# B&R Automation Studio project LMS47
Automation Studio 4.2.7.54 SP

## Configuration Config2

CPU 5PPC2100.BY22-000, AutomationRuntime B4.26, Build 4.1.2, Vc V4.26.2, Safety 0.0

### Task classes (Cpu.sw)
```
NcDataObjects: acp10etxen <- acp10etxen.dob, gAxis01i <- gAxis01obj.gAxis01i.dob, LMS47Liden <- gAxis01obj.LMS47Liden.dob
Libraries: Acp10man, Acp10par, NcGlobal, Acp10_MC, brsystem, sys_lib, runtime
```

### Hardware
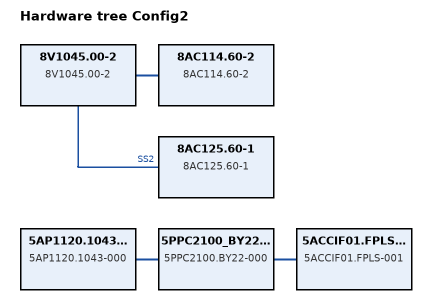
```
5ACCIF01.FPLS-001 : 5ACCIF01.FPLS-001 v1.2.0.0  [SL -> 5PPC2100_BY22_000b.SL1]
5AP1120.1043-000 : 5AP1120.1043-000 v1.0.1.0
5PPC2100_BY22_000b : 5PPC2100.BY22-000 v1.2.4.0  [SY -> 5AP1120.1043-000.SY1]
  Connector IF3:
    ActivateDevice = 1
  Connector IF4:
    ActivateDevice = 1
    Mode = Manual
    InternetAddress = 192.168.0.13
    SubnetMask = 255.255.255.0
  ConfigurationID = LMS47_Config2
  TimerDeviceType = EPLX2X
  TaskClassIdleTime = 2000
  Cyclic1Duration = 2000
  Cyclic1Tolerance = 0
  Cyclic2Duration = 20000
  Cyclic2Tolerance = 20000
  Cyclic3Duration = 50000
  Cyclic3Tolerance = 50000
  Cyclic4Duration = 100000
  Cyclic4Tolerance = 100000
  Cyclic5Duration = 200000
  Cyclic5Tolerance = 200000
  Cyclic6Duration = 500000
  Cyclic6Tolerance = 500000
  Cyclic7Duration = 1000000
  Cyclic7Tolerance = 1000000
  Cyclic8Duration = 10000
  Cyclic8Tolerance = 30000000
  TimerDevice = 5ACCIF01.FPLS-001.IF1
8AC114.60-2 : 8AC114.60-2 v1.0.0.8  [SS -> 8V1045.00-2.SS1; PLK1 -> 5ACCIF01.FPLS-001.IF1 (NodeNumber=1)]
8AC125.60-1 : 8AC125.60-1 v1.0.0.2  [SS -> 8V1045.00-2.SS2]
8V1045.00-2 : 8V1045.00-2 v1.0.0.2
  QuickStopIsNormallyOpen_r1 = on
```

### Acp10cfg.ncc - 5PPC2100_BY22_000b/Motion/Acp10cfg.ncc
```
NcConfiguration (Version=3.15.1, NcSwId=Acp10)
  ACP10CF1_typ:
    cnt_nettrc_rec_drive = 1500
    bufsize_trace_upload = 1200
    tc_nc_man_task = Cyclic #1
    glob_pv_as_ncobject = Yes
    ncsys_dl_broadcast = Yes
    ncsys_dl_acp_reset = Yes
    safemc_log_err_to_ax = Yes
    network_init:
      ncsw_init_execute = Yes
      automatic_execute = No
      node_nr_warning = Yes
      net_err_before_ncact = Yes
    nettrc:
      enter_parsecrec = Yes
      enter_ncaction = Yes
      save_ring_startidx = Yes
    cam_prof_download:
      cam_dat_dl_parallel = No
      tc_cam_dl_parallel = Task class for NC Manager task
    plk_if[0]:
      if_name = SL1.SS1.IF2
      tc_CycDat_PLCopen = Task class for NC Manager task
      mc_broadcast_extdat = No
    plk_if[1]:
      if_name = IF1
      tc_CycDat_PLCopen = Task class for NC Manager task
      mc_broadcast_extdat = No
    plk_if[2]:
      if_name = SL1.IF2
      tc_CycDat_PLCopen = Task class for NC Manager task
      mc_broadcast_extdat = No
    plk_if[3]:
      if_name = SL1.IF1
      tc_CycDat_PLCopen = Task class for NC Manager task
      mc_broadcast_extdat = No
```

### Acp10map.ncm - 5PPC2100_BY22_000b/Motion/Acp10map.ncm
```
NcMapping (NcSwId=Acp10, DisabledNodesAreHidden=False)
  NcObject gAxis01 (ModuleId=8V1045.00-2, Type=ncAXIS, Channel=1, AcoposSimulation=Off, InitParameter=gAxis01i, AcoposParameter=LMS47Liden, Disabled=FALSE, ModuleDisabled=FALSE)
  NcObject 8V1045.00-2_ncV_AXIS1 (ModuleId=8V1045.00-2, Type=ncV_AXIS, Channel=1, Disabled=TRUE, ModuleDisabled=FALSE)
```

## Logical view

Binary libraries used (declarations not repeated): operator, runtime, astime, AsIecCon, brsystem, sys_lib, Acp10man 3.15.1, Acp10par 3.15.1, NcGlobal 3.15.1, Acp10_MC 3.15.1

### Global.var - Global variables
```iecst
VAR
	gAxis01 : ACP10AXIS_typ;
	gAxSinCos : ACP10AXIS_typ;
	gAxis02 : ACP10AXIS_typ;
END_VAR
```


### Data object Logical/acp10etxen (Ett)

- acp10etxen.ett (not shown)

### Package Logical/gAxis01obj - gAxis01obj

### Data object Logical/gAxis01obj/LMS47Liden (Apt, version 1.00.0)

#### LMS47Liden.apt - rebuilt acopos parameter table (apt object) 
```
AcoposParameterTable:
  Root Parameters:
    Synchronous motor:
      General parameters:
        30 = 2 (Name=MOTOR_TYPE)  // Motor: Type
        31 = 513 (Name=MOTOR_COMPATIBILITY)  // Motor: Software compatibility
        46 = 1 (Name=MOTOR_WIND_CONNECT)  // Motor: Winding connection
        47 = 1 (Name=MOTOR_POLEPAIRS)  // Motor: Number of pole-pairs
      Brake parameters:
        42 = 0 (Name=MOTOR_BRAKE_CURR_RATED, Unit=A)  // Motor holding brake: Rated current
        43 = 0 (Name=MOTOR_BRAKE_TORQ_RATED, Unit=Nm)  // Motor holding brake: Rated torque
        44 = 0 (Name=MOTOR_BRAKE_ON_TIME, Unit=s)  // Motor holding brake: Engaging delay
        45 = 0 (Name=MOTOR_BRAKE_OFF_TIME, Unit=s)  // Motor holding brake: Release delay
      Thermo sensor parameters:
        64 = 0 (Name=MOTOR_TEMPSENS_PAR1)  // Temperature sensor: Parameter 1
        65 = 0 (Name=MOTOR_TEMPSENS_PAR2)  // Temperature sensor: Parameter 2
        66 = 0 (Name=MOTOR_TEMPSENS_PAR3)  // Temperature sensor: Parameter 3
        67 = 0 (Name=MOTOR_TEMPSENS_PAR4)  // Temperature sensor: Parameter 4
        68 = 0 (Name=MOTOR_TEMPSENS_PAR5)  // Temperature sensor: Parameter 5
        69 = 0 (Name=MOTOR_TEMPSENS_PAR6)  // Temperature sensor: Parameter 6
        70 = 0 (Name=MOTOR_TEMPSENS_PAR7)  // Temperature sensor: Parameter 7
        71 = 0 (Name=MOTOR_TEMPSENS_PAR8)  // Temperature sensor: Parameter 8
        72 = 0 (Name=MOTOR_TEMPSENS_PAR9)  // Temperature sensor: Parameter 9
        73 = 0 (Name=MOTOR_TEMPSENS_PAR10)  // Temperature sensor: Parameter 10
        75 = 0 (Name=MOTOR_THERMAL_CONST, Unit=s)  // Motor: Thermal time constant (for MOTOR_COMPATIBILITY 0x0202)
      Motor parameters:
        48 = 400 (Name=MOTOR_VOLTAGE_RATED, Unit=V)  // Motor: Rated voltage
        49 = 28.546301 (Name=MOTOR_VOLTAGE_CONST, Unit=mV*min)  // Motor: Voltage constant
        50 = 9375 (Name=MOTOR_SPEED_RATED, Unit=1/min)  // Motor: Rated speed
        51 = 18750 (Name=MOTOR_SPEED_MAX, Unit=1/min)  // Motor: Maximum speed
        52 = 3.73 (Name=MOTOR_TORQ_STALL, Unit=Nm)  // Motor: Stall torque
        53 = 3.73 (Name=MOTOR_TORQ_RATED, Unit=Nm)  // Motor: Rated torque
        54 = 7.4699998 (Name=MOTOR_TORQ_MAX, Unit=Nm)  // Motor: Peak torque
        55 = 0.47215188 (Name=MOTOR_TORQ_CONST, Unit=Nm/A)  // Motor: Torque constant
        56 = 7.9000001 (Name=MOTOR_CURR_STALL, Unit=A)  // Motor: Stall current
        57 = 7.9000001 (Name=MOTOR_CURR_RATED, Unit=A)  // Motor: Rated current
        58 = 23.700001 (Name=MOTOR_CURR_MAX, Unit=A)  // Motor: Peak current
        59 = 38.029545 (Name=MOTOR_WIND_CROSS_SECT, Unit=mmp)  // Motor: Phase cross section
        60 = 2.7743113 (Name=MOTOR_STATOR_RESISTANCE, Unit=Ohm)  // Motor: Stator resistance
        61 = 0.01827473 (Name=MOTOR_STATOR_INDUCTANCE, Unit=Henry)  // Motor: Stator inductance
        62 = 0.0020000001 (Name=MOTOR_INERTIA, Unit=kgmp)  // Motor: Moment of inertia
        63 = 1.1 (Name=MOTOR_COMMUT_OFFSET, Unit=rad)  // Motor: Commutation offset
        849 = 0 (Name=MOTOR_TAU_THERM, Unit=s)  // Motor: Thermal time constant
      Isolation parameters:
        74 = 120 (Name=MOTOR_WIND_TEMP_MAX, Unit=°C)  // Motor: Limit temperature
    Phasing:
      276 = 0 (Name=PHASING_MODE)  // Motor: Phasing: Mode
      275 = 13 (Name=PHASING_CURR, Unit=A)  // Motor: Phasing: Current
    BISS encoder (Disabled=FALSE)
      97 = ncBISS (Name=ENCOD_TYPE, Disabled=FALSE)  // Encoder1: Type
      109 = 32000 (Name=SCALE_ENCOD_INCR, Disabled=FALSE)  // Encoder1: Encoder scaling: increments per encoder revolution
      896 = 67 (Name=ENCOD_CRC_POLYNOMIAL, Disabled=FALSE)  // Encoder1: CRC Polynomial
      1370 = 0 (Name=ENCOD_SSI_CONTENT_IDX, Disabled=FALSE)  // Encoder1: SSI content index
      1371 = ncSSI_CONT_TYP_POS (Name=ENCOD_SSI_CONTENT_TYPE, Disabled=FALSE)  // Encoder1: SSI content type
      238 = 32 (Name=ENCOD_SSI_BITS, Disabled=FALSE)  // Encoder1: SSI Number of data bits
      1370 = 1 (Name=ENCOD_SSI_CONTENT_IDX, Disabled=FALSE)  // Encoder1: SSI content index
      1371 = ncSSI_CONT_TYP_ERR_INV (Name=ENCOD_SSI_CONTENT_TYPE, Disabled=FALSE)  // Encoder1: SSI content type
      238 = 1 (Name=ENCOD_SSI_BITS, Disabled=FALSE)  // Encoder1: SSI Number of data bits
      1370 = 2 (Name=ENCOD_SSI_CONTENT_IDX, Disabled=FALSE)  // Encoder1: SSI content index
      1371 = ncSSI_CONT_TYP_FILL (Name=ENCOD_SSI_CONTENT_TYPE, Disabled=FALSE)  // Encoder1: SSI content type
      238 = 1 (Name=ENCOD_SSI_BITS, Disabled=FALSE)  // Encoder1: SSI Number of data bits
      1370 = 3 (Name=ENCOD_SSI_CONTENT_IDX, Disabled=FALSE)  // Encoder1: SSI content index
      1371 = ncSSI_CONT_TYP_END (Name=ENCOD_SSI_CONTENT_TYPE, Disabled=FALSE)  // Encoder1: SSI content type
    347 = 10000 (Name=F_SWITCH, Unit=cps, Disabled=TRUE)  // Inverter: Switch frequency
```

### Data object Logical/gAxis01obj/gAxis01i (Ax)

#### gAxis01i.ax
```
InitParameter (Version=3.15.1, NcSwId=ACP10)
  ACP10AXIS_typ:
    dig_in:
      level:
        reference = ncACTIV_LO
        pos_hw_end = ncACTIV_HI
        neg_hw_end = ncACTIV_HI
        trigger1 = ncACTIV_HI
        trigger2 = ncACTIV_HI
    encoder_if:
      parameter:
        count_dir = ncSTANDARD
        scaling:
          load:
            units = 32000
            rev_motor = 1
    limit:
      parameter:
        v_pos = 1.0E+07
        v_neg = 1.0E+07
        a1_pos = 3.0E+07
        a2_pos = 3.0E+07
        a1_neg = 3.0E+07
        a2_neg = 3.0E+07
        t_jolt = 0.03
        t_in_pos = 0.0
        pos_sw_end = 620000
        neg_sw_end = 5000
        ds_warning = 1000.0
        ds_stop = 1000.0
        a_stop = 1.0E+30
        dv_stop = 0.0
        dv_stop_mode = ncOFF
    controller:
      mode = ncPOSITION + ncFF
      position:
        kv = 275.9
        tn = 0.0
        t_predict = 0.0004
        t_total = 0.0004
        p_max = 1.0E+30
        i_max = 0.0
      speed:
        kv = 7.55
        tn = 0.0
        t_filter = 0.0004
        isq_filter1:
          type = ncOFF
          a0 = 0.0
          a1 = 0.0
          b0 = 0.0
          b1 = 0.0
          b2 = 0.0
          c0_par_id = 0
          c1_par_id = 0
        isq_filter2:
          type = ncOFF
          a0 = 0.0
          a1 = 0.0
          b0 = 0.0
          b1 = 0.0
          b2 = 0.0
          c0_par_id = 0
          c1_par_id = 0
        isq_filter3:
          type = ncOFF
          a0 = 0.0
          a1 = 0.0
          b0 = 0.0
          b1 = 0.0
          b2 = 0.0
          c0_par_id = 0
          c1_par_id = 0
      uf:
        type = ncLINEAR
        auto_config = ncMOTOR_PAR
        u0 = 0.0
        un = 0.0
        fn = 50.0
        k_f_slip = 0.0
      ff:
        torque_load = 0.0
        torque_pos = 0.201724
        torque_neg = 0.166364
        kv_torque = 0.0266516
        inertia = 0.00166562
        t_filter_a = 0.0
    move:
      stop:
        parameter[0]:
          decel_ramp = ncA_LIMIT
          controller = ncON
        parameter[1]:
          decel_ramp = ncA_LIMIT
          controller = ncON
        parameter[2]:
          decel_ramp = ncA_LIMIT
          controller = ncON
        parameter[3]:
          decel_ramp = ncA_LIMIT
          controller = ncON
        quickstop:
          decel_ramp = ncA_LIMIT
        drive_error:
          decel_ramp = ncA_LIMIT
      homing:
        parameter:
          s = 0
          v_switch = 5000.0
          v_trigger = 500.0
          a = 50000.0
          mode = ncDIRECT
          edge_sw = ncPOSITIVE
          start_dir = ncPOSITIVE
          trigg_dir = ncPOSITIVE
          ref_pulse = ncOFF
          fix_dir = ncOFF
          tr_s_block = 0.0
          torque_lim = 0.0
          ds_block = 0.0
          ds_stop = 0.0
      basis:
        parameter:
          v_pos = 3000000.0
          v_neg = 3000000.0
          a1_pos = 1.6E+07
          a2_pos = 1.6E+07
          a1_neg = 1.6E+07
          a2_neg = 1.6E+07
    message:
      text:
        parameter:
          format = ncBREAK
          columns = 80
          data_modul = acp10etxen
```

Listed in the project but not available here: Logical/Global.typ
